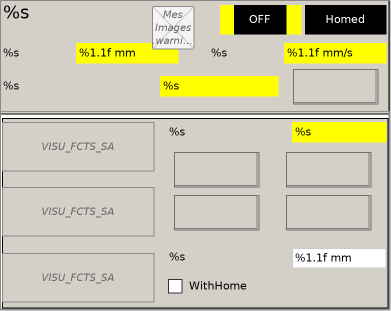
VISUALIZATION VISU_CANNE_TRANSFERT  // 391x311
VAR_IN_OUT
	m_Input_Moteur:				BLOCK_AXE_STD1;
	m_Input_Id_Poste:			INT;
	m_Input_Command_Visible:	BOOL;	
END_VAR
    Rectangle (0,0 389x114), "%s", text list: 'TextList_Canne_Transfert', text index: 0
    RoundedRectangle (220,5 81x29), invisible if: NOT m_Input_Moteur.OP_Validation.AR
    RoundedRectangle (220,5 81x29), invisible if: NOT m_Input_Moteur.OP_Validation.OK
    RoundedRectangle (220,5 81x29), invisible if: NOT m_Input_Moteur.OP_Validation.EC
    RoundedRectangle (234,5 52x29), "ON", invisible if: m_Input_Moteur.STATE_Ar
    RoundedRectangle (234,5 52x29), "OFF", invisible if: NOT m_Input_Moteur.STATE_Ar
    RoundedRectangle (305,5 81x29), "Homed", invisible if: NOT m_Input_Moteur.STATE_Homed OR m_Input_Moteur.CONF_No_Ref
    RoundedRectangle (305,5 81x29), "Homed", invisible if: m_Input_Moteur.STATE_Homed OR m_Input_Moteur.CONF_No_Ref
    Textfield (0,43 120x20), "%s", text list: 'TextList_Canne_Transfert', text index: 1
    Textfield (76,43 102x20), "%1.1f mm", text variable: m_Input_Moteur.STATE_Pos
    Textfield (208,43 120x20), "%s", text list: 'TextList_Canne_Transfert', text index: 2
    Textfield (284,43 102x20), "%1.1f mm/s", text variable: m_Input_Moteur.STATE_Vit
    Textfield (0,76 153x20), "%s", text list: 'TextList_Canne_Transfert', text index: 3
    Textfield (160,76 118x20), "%s", text list: 'TextList_Position_Canne', text index: m_Input_Id_Poste
    GroupBox (0,103 389x206), invisible if: NOT m_Input_Command_Visible
        Rectangle (2,15 386x190)
        Frame (2,19 152x49)
            shows VISU_FCTS_SA(m_Input_ID_XML := 6, m_Input_UserRight := PRG_USER.ACTU_USER.FONCTION_SA, m_Input_Operation := m_Input_Moteur.OP_Validation)
        Frame (2,150 152x49)
            shows VISU_FCTS_SA(m_Input_ID_XML := 8, m_Input_UserRight := PRG_USER.ACTU_USER.FONCTION_SA, m_Input_Operation := m_Input_Moteur.OP_Position)
        Frame (2,84 152x49)
            shows VISU_FCTS_SA(m_Input_ID_XML := 7, m_Input_UserRight := PRG_USER.ACTU_USER.FONCTION_SA, m_Input_Operation := m_Input_Moteur.OP_Stop)
        Checkbox (166,171 145x24), "WithHome", variable: m_Input_Moteur.PRM_GoToHome
        Textfield (166,19 120x20), "%s", text list: 'TextList_Canne_Transfert', text index: 4
        Textfield (292,19 94x20), "%s", text list: 'TextList_Position_Canne', text index: m_Input_Moteur.PRM_NRef
        Button (174,49 85x35), input disabled if: NOT PRG_USER.ACTU_USER.FONCTION_SA, text list: 'TextList_Position_Canne', text index: 0
            OnMouseClick: execute { m_Input_Moteur.PRM_NREF := 0; }
        Button (286,49 85x35), input disabled if: NOT PRG_USER.ACTU_USER.FONCTION_SA, text list: 'TextList_Position_Canne', text index: 1
            OnMouseClick: execute { m_Input_Moteur.PRM_NREF := 1; }
        Button (174,92 85x35), input disabled if: NOT PRG_USER.ACTU_USER.FONCTION_SA, text list: 'TextList_Position_Canne', text index: 2
            OnMouseClick: execute { m_Input_Moteur.PRM_NREF := 2; }
        Textfield (166,144 120x20), "%s", text list: 'TextList_Canne_Transfert', text index: 5
        Textfield (292,145 94x20), "%1.1f mm", text variable: m_Input_Moteur.PRM_Position
            OnMouseClick: write the text variable via VisuDialogs.NumpadExtended, min -100, max 100
        Button (286,92 85x35), input disabled if: NOT PRG_USER.ACTU_USER.FONCTION_SA, text list: 'TextList_Position_Canne', text index: 3
            OnMouseClick: execute { m_Input_Moteur.PRM_NREF := 3; }
    Button (293,69 85x35), text list: 'TextList_Canne_Transfert', text index: 7
        toggle m_Input_Command_Visible
    Image (152,6 42x43), invisible if: NOT m_Input_Moteur.STATE_NOK, image: MesImages.warning
END_VISUALIZATION

(* stored: Version 1.1.0.1, ProductVersion 3.1.4024.10
   Visu VISU_CANNE_TRANSFERT: Id {4187b5e3-ef2e-40d4-818a-e35c9fe9404b} *)
